// TwinCAT 3 PLC project Aufgabensammlung2
// ProgramVersion: 3.1.4023.0
// libraries:
//   Tc2_Standard, * (Beckhoff Automation GmbH)
//   Tc2_System, * (Beckhoff Automation GmbH)
//   Tc3_Module, * (Beckhoff Automation GmbH)
// project tree:
//   / PlcTask.TcTTO
//   POUs/ DoSomeMath.TcPOU, fb_Counter.TcPOU, fb_test.TcPOU, f_Addition.TcPOU, f_Division.TcPOU, f_Subtraction.TcPOU, MAIN.TcPOU, f_Multiplication.TcPOU
// real-time tasks:
//   TASK PlcTask: cycle T#10ms, priority 20, ADS port 350
//   TASK PlcTask1: cycle T#10ms, priority 21, ADS port 351

CONFIGURATION Aufgabensammlung2
    RESOURCE PLC ON TwinCAT3
        TASK PlcTask(INTERVAL := T#10ms, PRIORITY := 20);
        PROGRAM MAIN WITH PlcTask : MAIN;
    END_RESOURCE
END_CONFIGURATION

// ---- POUs/MAIN.TcPOU
PROGRAM MAIN
VAR
	FBCounter	: fb_Counter;
	iZaehler	: INT := 0;
END_VAR

// Aufrufmöglichkeit 1
FBCounter.bActive	:= TRUE;
FBCounter.bReset	:= FALSE;
FBCounter();
iZaehler := FBCounter.iCounter;
// Aufrufmöglichkeit 2
FBCounter(bActive := TRUE, bReset := FALSE, iCounter=>iZaehler);

END_PROGRAM

// ---- POUs/fb_Counter.TcPOU
FUNCTION_BLOCK fb_Counter
VAR_INPUT
	bActive		:	BOOL;
	bReset		:	BOOL;
END_VAR
VAR_OUTPUT
	iCounter	:	INT;
END_VAR
VAR
END_VAR

IF bActive THEN
	iCounter := iCounter + 1;
ELSE
	IF bReset THEN
		iCounter := 0;
	END_IF
END_IF

END_FUNCTION_BLOCK

// ---- POUs/DoSomeMath.TcPOU
PROGRAM DoSomeMath
VAR
	rValue1	: REAL	:= 7;	
	rValue2	: REAL	:= 2;
	rResult	: REAL	:= 0;
	
	iCounter : INT := 0;
	
	//Test Array
	aTestArray 	: ARRAY[0..10] OF INT;
	iTestValue	: INT := 0;
	
END_VAR

rResult := f_Addition(rSum1 := rValue1, rSum2 := rValue2);
rResult := f_Multiplication(rValue1, rValue2);
rResult := f_Division(aTestArray[2], rValue2);
iCounter := iCounter + 1;

FOR iTestValue := 0 TO 10 BY 1 DO
	aTestArray[iTestValue] := iCounter;
	 IF iTestValue >3 THEN
		 EXIT;
	 END_IF
END_FOR

END_PROGRAM

// ---- POUs/f_Addition.TcPOU
FUNCTION f_Addition : REAL
VAR_INPUT
	rSum1	:	REAL;
	rSum2	:	REAL;
END_VAR
VAR
END_VAR

f_Addition := rSum1 + rSum2;

END_FUNCTION

// ---- POUs/f_Multiplication.TcPOU
FUNCTION f_Multiplication : REAL
VAR_INPUT
	rProd1	:	REAL;
	rProd2	:	REAL;
END_VAR
VAR
END_VAR

f_Multiplication := rProd1	* rProd2;

END_FUNCTION

// ---- POUs/f_Division.TcPOU
FUNCTION f_Division : REAL
VAR_INPUT
	rDiv	:	REAL;
	rQout	:	REAL;
END_VAR
VAR
END_VAR

IF  rQout = 0 THEN
	f_Division := 0;
ELSE
	f_Division := rDiv / rQout;
END_IF

END_FUNCTION

// ---- POUs/fb_test.TcPOU
FUNCTION_BLOCK fb_test
VAR_INPUT
END_VAR
VAR_OUTPUT
END_VAR
VAR
END_VAR

END_FUNCTION_BLOCK

// ---- POUs/f_Subtraction.TcPOU
FUNCTION f_Subtraction : REAL
VAR_INPUT
	rDiff1	:	REAL;
	rDiff2	:	REAL;
END_VAR
VAR
END_VAR

f_Subtraction := rDiff1 - rDiff2;

END_FUNCTION
